/// `TcLogCore` provides the base functionality of the logger and sets the configuration.
/// The logger can be configured by calling its methods that set the configuration.
///
/// > [!NOTE]
/// > `TcLogCore.RunLogger()` should be called once each cycle. The configuration methods should be called **before** 
/// > `RunLogger` is called.
///
/// When declaring an instance of TcLogCore, the ininital buffer size has to be set. If the buffer size is set too low, it will expand
/// automatically if enough memory is available.
///
/// To set the inital buffer size to accomodate 100 messages, use it like this:
///
/// ```st
/// VAR
///   myLogger: TcLogCore(BufferSize := 100 * (Tc2_System.MAX_STRING_LENGTH * Constants.FifoOverhead));
/// END_VAR
/// ```
///
{attribute 'linkalways'} 
{attribute 'no_explicit_call' := 'This FB is a CLASS and must be accessed using methods or properties'}
{attribute 'enable_dynamic_creation'}
{attribute 'hide_all_locals'}
FUNCTION_BLOCK TcLogCore IMPLEMENTS LogCore
VAR
	logging_singleton : TcLog; // Logger-Singleton: Required to provide Singleton-functionality for TcLog.
	utc_time_as_file_time : Tc2_Utilities.T_FileTime; // Current utc time as filetime
	local_time_as_system_time : Tc2_Utilities.TimeStruct; // Current local time as timestring
	local_time_as_string : STRING; // Current local time as string
	log_cache : DynamicStringBuffer; // Dynamic string buffer to cache logs to be processed
	start_logging_configuration : BOOL; // Aux variable to provide fluent interface.
	internal_error_occured : BOOL; // Aux variable to log internal errors to Error-property.                                                   				
	_config : LoggingConfiguration; // Logging configuration. Is set by invoking configuration methods.
	_error : Error; // Contains information about internal error.
	_busy : BOOL; // Logger is busy, typically with writing logs to the file system.
	time_info_ready : BOOL := FALSE; // Set to true once the time information is available
END_VAR

// Nothing to be done here. Logger works by invoking its methods.
// "RunLogger" contains all the implementation that has to be processed cyclically.

// Builds logging configuration.
// Required to provide a fluent interface.
// Has to be called at the begin of each method that configures the logger.
{attribute 'hide'}
METHOD PRIVATE BuildLoggingConfiguration : BOOL
IF NOT start_logging_configuration THEN
	start_logging_configuration := TRUE;
	
	_config.rolling_interval := RollingIntervals.Daily;
	_config.write_to_ads := FALSE;
	_config.file_name := '';
	_config.file_path := 'c:\';
	_config.minimum_level := LogLevel.Debug;
	_config.delimiter := '|';
	_config.include_instance_path := FALSE;
	_config.log_file_life_span := 0;
	_config.timestamp_format := 'YYYYMMDD_hhmm_';
	_config.valid_timestamps_only := FALSE;
END_IF
END_METHOD

/// `Busy` evaluates to `TRUE` as long as the log file is kept open to append new log messages
/// or there are pending messages in the queue to be written to the logfile.
{attribute 'monitoring':='call'}
PROPERTY Busy : BOOL
GET
Busy := _busy;
END_GET
SET // PRIVATE
_busy := Busy;
END_SET
END_PROPERTY

/// Returns the current configuration of the logger.
{attribute 'monitoring':='variable'}
PROPERTY Configuration : LoggingConfiguration
GET
Configuration := _config;
END_GET
END_PROPERTY

/// Configuration method which sets the lifespan of log files. Once exceeded, they will be deleted.
METHOD DeleteLogFilesAfterDays : REFERENCE TO TcLogCore
VAR_INPUT
  /// Lifespan of logfiles in days.
	lifespan : UINT; 
END_VAR
BuildLoggingConfiguration();

_config.log_file_life_span := lifespan;

DeleteLogFilesAfterDays REF= THIS^;
END_METHOD

/// Returns information about internal errors.
{attribute 'monitoring':='call'}
{attribute 'suppress_wrn_C0410'}
PROPERTY Error : REFERENCE TO Error
GET
Error REF= _error;
END_GET
END_PROPERTY

METHOD FB_init : BOOL
VAR_INPUT
	bInitRetains : BOOL; // if TRUE, the retain variables are initialized (warm start / cold start)
	bInCopyCode : BOOL; // if TRUE, the instance afterwards gets moved into the copy code (online change)
	/// Initial buffer size for the internal log message buffer
	bufferSize : UDINT;
END_VAR
logging_singleton.Init(THIS^);
log_cache.Init(bufferSize);
END_METHOD

/// Flushes the logging cache. All messages that have not yet been processed will be lost.
METHOD FlushCache : BOOL
log_cache.FlushCache();
END_METHOD

/// Configuration method. If this method is called, the instance path where the log 
/// messages has been triggered will be included in the log message. 
METHOD IncludeInstancePath : REFERENCE TO TcLogCore
BuildLoggingConfiguration();

_config.include_instance_path := TRUE;

IncludeInstancePath REF= This^;
END_METHOD

/// Logger method. It should only be called from within objects that implement `ILog`.
/// Logs data in custom format. No additional formatting will be done. 
METHOD LogCustomFormat : BOOL
VAR_INPUT
	/// Data to be logged.
	data : Tc2_System.T_MaxString; 
END_VAR
IF(TimeInfoReady OR NOT _config.valid_timestamps_only) THEN 
	IF _config.write_to_ads THEN 
		Tc2_System.AdsLogStr(Tc2_System.AdsLog_MsgType_Log OR Tc2_System.AdsLog_MsgType_Hint, data, ''); 
	END_IF
	
	IF _config.file_name <> '' THEN 
		log_cache.AddLine(data);
	END_IF
END_IF
END_METHOD

/// Logger method. It should only be called from within objects that implement `ILog`.
/// Logs in the standard format. This includes
/// - timestamp
/// - log level
/// - log message
/// - instance path of logging source (optional)
/// The message will only be logged if the logging level exceeds the configured minimum logging level.
METHOD LogStandardFormat : BOOL
VAR_INPUT
  /// Data to be logged.
	data : Tc2_System.T_MaxString; 
  /// Instance path of calling logger to locate source of logging message.
	instance_path : Tc2_System.T_MaxString;
  /// Log level of message. 
	log_level : LogLevel; 
END_VAR
VAR_INST
  {attribute 'hide'}
	message_builder : DefaultStringBuilder;
END_VAR
IF log_level >= _config.minimum_level AND (TimeInfoReady OR NOT _config.valid_timestamps_only)  THEN
	IF _config.write_to_ads THEN 
		Tc2_System.ADSLOGSTR(
			Tc2_System.AdsLog_MsgType_Log OR LogLevelToAdsLogMsgType(log_level), 
			message_builder
				.Reset()
				.AppendIf(_config.include_instance_path, instance_path)
				.AppendIf(_config.include_instance_path, _config.delimiter)
				.Append(data)
				.ToString(), 
			''
		); 
	END_IF
	
	IF _config.file_name <> '' THEN 
		log_cache.AddLine(
			message_builder
					.Reset()
					.Append(local_time_as_string)
					.Append(_config.delimiter)
					.Append(TO_STRING(log_level))
					.AppendIf(_config.include_instance_path, _config.delimiter)
					.AppendIf(_config.include_instance_path, instance_path)
					.Append(_config.delimiter)
					.Append(data)
					.ToString()
		);
	END_IF
END_IF
END_METHOD

/// Logger method. Structured attributes are currently discarded by this backend.
/// A future WriteToJsonFile configuration method can use attrs/attr_count here.
METHOD LogWithAttributes : BOOL
VAR_INPUT
    data : Tc2_System.T_MaxString;
    instance_path : Tc2_System.T_MaxString;
    log_level : LogLevel;
    attrs : ARRAY[0..9] OF LogAttribute;
    attr_count : USINT;
END_VAR
// Delegate to existing standard-format logic — attributes are discarded by this backend.
LogWithAttributes := LogStandardFormat(data, instance_path, log_level);
END_METHOD

/// Configuration method.
/// Sets the minimum log level. Log messages below this level 
/// will not be logged.
METHOD MinimumLevel : REFERENCE TO TcLogCore
VAR_INPUT
  /// Minimum log level to be logged.
	level : LogLevel; 
END_VAR
BuildLoggingConfiguration();

_config.minimum_level := level;

MinimumLevel REF=THIS^;
END_METHOD

// Checks the specified rolling interval for the file name.
// Generates new file name if rolling intervall exceeded.
{attribute 'hide_all_locals'}
{attribute 'hide'}
METHOD PRIVATE RollingIntervalReached : BOOL
VAR_INPUT
	currentUtcTime : Tc2_Utilities.TIMESTRUCT;  // Current system time as utc
	rollingInterval : RollingIntervals; // Rolling interval 
END_VAR
VAR_INST
	newHour : Tc2_Standard.R_TRIG;
	newDay : Tc2_Standard.R_TRIG;
	newMonth : Tc2_Standard.R_TRIG;
	
	hourRolled : BOOL;
	dayRolled : BOOL;
	monthRolled : BOOL;
END_VAR
newHour(CLK := (currentUtcTime.wMinute = 0 AND currentUtcTime.wSecond = 0), 
	Q => hourRolled);
newDay(CLK := (hourRolled AND currentUtcTime.wHour = 0), 
	Q => dayRolled);
newMonth(CLK := (dayRolled AND currentUtcTime.wDay = 1), 
	Q => monthRolled);

RollingIntervalReached := 	(hourRolled 	AND rollingInterval = RollingIntervals.Hourly) OR
							(dayRolled 		AND rollingInterval = RollingIntervals.Daily) 	OR
							(monthRolled 	AND rollingInterval = RollingIntervals.Monthly);
END_METHOD

/// Cyclic method of Logger.
/// This method has to be executed in every plc cycle and runs 
/// all internal methods that have to be executed cyclically.
/// > [!NOTE]
/// > This method should be the last method of `TcLogCore` to be called in each cycle.
{attribute 'hide_all_locals'}
METHOD RunLogger : BOOL
VAR_INST
	new_day : Tc2_Standard.R_Trig; 
	dateTime : DateTime;
	delete_expired_log_files : DeleteOldFiles;
	file_name_string_builder : DefaultStringBuilder;
	timestamp : STRING; // Timestamp used for filename
END_VAR
// Generate time data (shared state)
dateTime();
IF dateTime.Done THEN time_info_ready := TRUE; END_IF

local_time_as_system_time := dateTime.AsLocalSystemTime;
local_time_as_string := dateTime.AsLocalSystemTimeString;
utc_time_as_file_time := dateTime.AsUtcFileTime;

// Generate new timestamp for filename
IF RollingIntervalReached(local_time_as_system_time, _config.rolling_interval) OR dateTime.Done THEN
	timestamp := dateTime.ToFormatString(_config.timestamp_format);
END_IF

// Delete expired log files
new_day(CLK := local_time_as_system_time.wHour = 0);
delete_expired_log_files(
	StartScan := 	new_day.Q AND (_config.log_file_life_span > 0),
	ExpirationInDays :=	_config.log_file_life_span,
	FilePath :=	_config.file_path,
	FileName :=	_config.file_name,
	current_utc_time := 	utc_time_as_file_time	
	);
IF delete_expired_log_files.Error.Active THEN
	internal_error_occured := TRUE;
	_error := delete_expired_log_files.Error;
END_IF
		
// Persist logging messages to file
log_cache.PersistToFile(
  TimeInfoReady,
	file_name_string_builder
		.Reset()
		.Append(_config.file_path)
		.AppendIf(Tc2_Standard.RIGHT(_config.file_path, 1) <> '\', '\')
		.Append(timestamp)
		.Append(_config.file_name)
		.ToString()
);
IF log_cache.Error.Active THEN
	internal_error_occured := TRUE;
	_error := log_cache.Error;
END_IF

// Forward busy state of LogCache 
Busy := log_cache.Busy;

// Reset Logging configuration: neccesary in order to provide fluent interface
start_logging_configuration := FALSE;

// Reset error flag each cycle to automatically confirm errors once they are gone.
IF NOT internal_error_occured THEN
	_error.Active := FALSE;
	_error.Code := ErrorCodes.None;
	_error.Info := '';
END_IF
internal_error_occured := FALSE;
END_METHOD

/// Configuration method
/// Sets delimiter between different columns of log file.
METHOD SetDelimiter : REFERENCE TO TcLogCore
VAR_INPUT
  /// Delimiter between different columns of log file.
	delimiter : STRING(1); 
END_VAR
BuildLoggingConfiguration();

_config.delimiter := delimiter;

SetDelimiter REF=THIS^;
END_METHOD

/// Configuration method.
/// Sets the rolling interval of the log file. Once the rolling interval
/// expires, a file name with a new timestamp will be generated.
METHOD SetRollingInterval : REFERENCE TO TcLogCore
VAR_INPUT
  /// Rolling interval for log file. Once exceeded, a new log file will be created.
	interval : RollingIntervals; 
END_VAR
BuildLoggingConfiguration();

_config.rolling_interval := interval;

SetRollingInterval REF= THIS^;
END_METHOD

/// `TimeInfoReady` evaluates to `TRUE` once the time information used by determine
/// the timestamp for the message is available.
{attribute 'monitoring':='call'}
PROPERTY TimeInfoReady : BOOL
GET
TimeInfoReady := time_info_ready;
END_GET
END_PROPERTY

/// Configuration method.
/// Sets the format of the timestamp in the file name. 
/// 
/// The following format options are available:
///	Y : year
///	M : month
/// D : day
/// h : hour 
/// m : minute
/// s : second
/// i : millisecond
/// 
/// Example: _YYMMDD-hh:mm:ss:iii_
/// => _20210812-12:30:22:123_
METHOD TimestampFormat : REFERENCE TO TcLogCore
VAR_INPUT
  /// Format the timestamp should have.
	format : STRING; 
END_VAR
BuildLoggingConfiguration();

_config.timestamp_format := format;

TimestampFormat REF= THIS^;
END_METHOD

/// Configuration method. If this method is called, only valid timestamps are logged.
/// Note that using this configuration will skip logging anything during the first few PLC cycles, 
/// as TwinCAT needs a few cycles to initialize its time information.
METHOD ValidTimestampsOnly : REFERENCE TO TcLogCore
BuildLoggingConfiguration();

_config.valid_timestamps_only := TRUE;

ValidTimestampsOnly REF= This^;
END_METHOD

/// Configuration method.
/// If this method is called, the logs will be written to ADS.
METHOD WriteToAds : REFERENCE TO TcLogCore
BuildLoggingConfiguration();

_config.write_to_ads := TRUE;

WriteToAds REF= This^;
END_METHOD

/// Configuration method.
/// If this method is called, the logs will be persisted to the file system.
METHOD WriteToFile : REFERENCE TO TcLogCore
VAR_INPUT
	/// File path the logs will be written to.
	path : Tc2_System.T_MaxString; 
	/// File name of the log file. Will automatically be prefixed by timestamp.
	file_name : STRING; 
END_VAR
BuildLoggingConfiguration();

IF Tc2_Standard.RIGHT(path, 1) <> '\' THEN
	_config.file_path := TC2_Standard.CONCAT(path, '\');  
ELSE
	_config.file_path := path;
END_IF
_config.file_name := file_name;

WriteToFile REF= This^;
END_METHOD

END_FUNCTION_BLOCK

(* stored: Version 1.1.0.1
   POU TcLogCore: Id {36505e85-a5ae-4de1-9bf6-165bd9e8fb7c}, SpecialFunc None
   Method BuildLoggingConfiguration: Id {414139bc-5769-4963-8989-c84f471a88a9}
   Property Busy: Id {8f16f6a4-6d8a-4697-8588-979372ae7eee}
   Get Get: Id {417d4c3d-9a0b-40e7-be03-0311ddfb3e62}
   Set Set: Id {704a377a-34a4-4b7b-ae17-6ec4a001a613}
   Property Configuration: Id {b69ecf4e-c3e0-42b6-9a58-14d24f318318}
   Get Get: Id {336f3bb8-888c-4134-9f52-f32abb54806d}
   Method DeleteLogFilesAfterDays: Id {3f478fd2-c36f-4c8d-ac26-2e0e30dfcf3f}
   Property Error: Id {07eb83c0-170b-480f-8f22-5aef3ef9c3c2}
   Get Get: Id {e0cb0c8f-130e-4ce7-9ace-bf920ab0cf4d}
   Method FB_init: Id {623ef1bb-99a1-4c18-a6cc-144772106b6d}
   Method FlushCache: Id {c8fe275e-8220-467f-9357-393f375a5ed5}
   Method IncludeInstancePath: Id {ccd76952-cda0-42c9-9588-571441e573a8}
   Method LogCustomFormat: Id {f6452548-6bc2-47c8-95b8-3de75137dfb8}
   Method LogStandardFormat: Id {d655b0a4-8e07-4fda-a759-8f830843bfc5}
   Method LogWithAttributes: Id {3792088f-e537-42fd-97cc-8dfa095a346c}
   Method MinimumLevel: Id {bebb146b-3a3d-45ce-aa61-48ddc123e45d}
   Method RollingIntervalReached: Id {5bc9e8c4-87c9-4c47-988c-39d834e79ac0}
   Method RunLogger: Id {bd6bd51f-2e6e-4802-b52c-34c2635bc527}
   Method SetDelimiter: Id {ae68ab0e-2db1-437e-bc56-0129dc5c983f}
   Method SetRollingInterval: Id {2a5a17a6-99f2-4763-b1c1-52b694f8f1e1}
   Property TimeInfoReady: Id {84ad0941-65a4-4e7b-8427-bb17b37f5fe5}
   Get Get: Id {52c72a65-8a03-4c7e-9ab8-7b61c68dec66}
   Method TimestampFormat: Id {f91c7e6e-6b5a-4b12-8b6e-be3f35191376}
   Method ValidTimestampsOnly: Id {7b350e30-415f-46a9-b7ed-d8ad47818f5f}
   Method WriteToAds: Id {f7faaafa-a500-40f8-aebf-2407a34de80e}
   Method WriteToFile: Id {084bec22-7d00-4dd8-a2b0-7bbb126ebf3c} *)
